// TIA Portal V20 export
FUNCTION "RealFcName" : Void   // FC1, LAD
   VAR_INPUT
      Input : Real;
   END_VAR
   VAR_OUTPUT
      Output : Real;
   END_VAR
BEGIN
END_FUNCTION
